PROGRAM AxisStop
VAR	
	
END_VAR

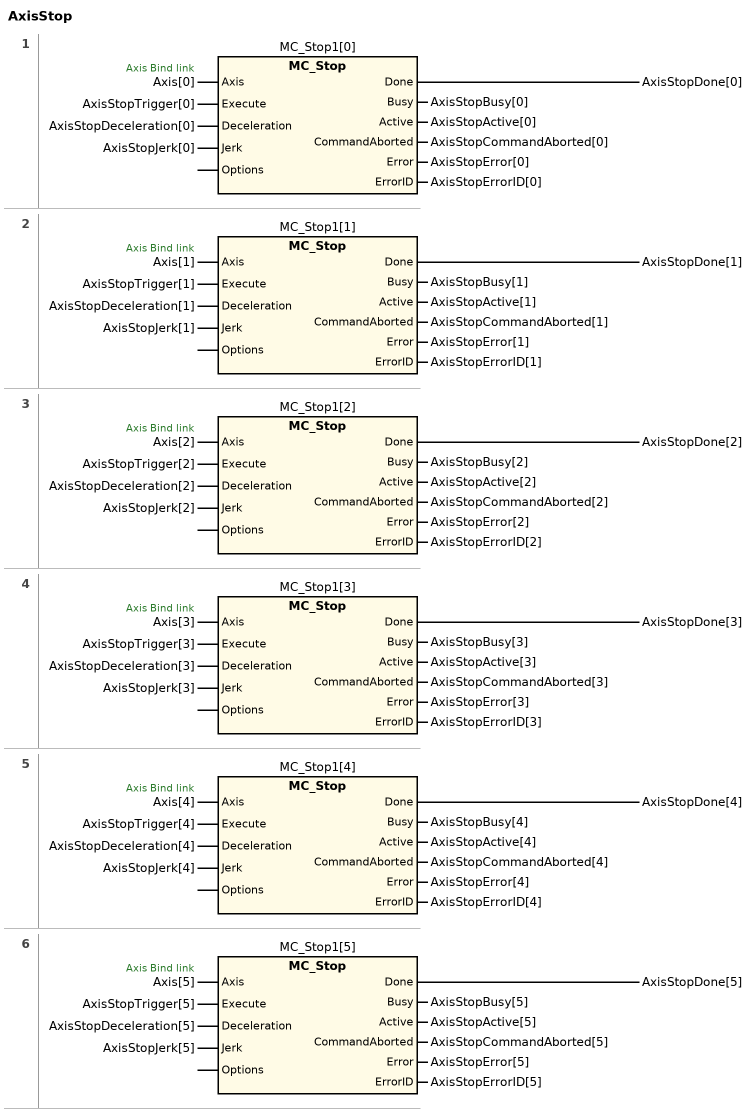
// NETWORK 1
//   MC_Stop1[0]: Axis Stop
//   Axis[0]: Axis Bind link
MC_Stop1[0](
    Axis := Axis[0],
    Execute := AxisStopTrigger[0],
    Deceleration := AxisStopDeceleration[0],
    Jerk := AxisStopJerk[0],
    Busy => AxisStopBusy[0],
    Active => AxisStopActive[0],
    CommandAborted => AxisStopCommandAborted[0],
    Error => AxisStopError[0],
    ErrorID => AxisStopErrorID[0]); // MC_Stop
AxisStopDone[0] := MC_Stop1[0].Done;

// NETWORK 2
//   MC_Stop1[1]: Axis Stop
//   Axis[1]: Axis Bind link
MC_Stop1[1](
    Axis := Axis[1],
    Execute := AxisStopTrigger[1],
    Deceleration := AxisStopDeceleration[1],
    Jerk := AxisStopJerk[1],
    Busy => AxisStopBusy[1],
    Active => AxisStopActive[1],
    CommandAborted => AxisStopCommandAborted[1],
    Error => AxisStopError[1],
    ErrorID => AxisStopErrorID[1]); // MC_Stop
AxisStopDone[1] := MC_Stop1[1].Done;

// NETWORK 3
//   MC_Stop1[2]: Axis Stop
//   Axis[2]: Axis Bind link
MC_Stop1[2](
    Axis := Axis[2],
    Execute := AxisStopTrigger[2],
    Deceleration := AxisStopDeceleration[2],
    Jerk := AxisStopJerk[2],
    Busy => AxisStopBusy[2],
    Active => AxisStopActive[2],
    CommandAborted => AxisStopCommandAborted[2],
    Error => AxisStopError[2],
    ErrorID => AxisStopErrorID[2]); // MC_Stop
AxisStopDone[2] := MC_Stop1[2].Done;

// NETWORK 4
//   MC_Stop1[3]: Axis Stop
//   Axis[3]: Axis Bind link
MC_Stop1[3](
    Axis := Axis[3],
    Execute := AxisStopTrigger[3],
    Deceleration := AxisStopDeceleration[3],
    Jerk := AxisStopJerk[3],
    Busy => AxisStopBusy[3],
    Active => AxisStopActive[3],
    CommandAborted => AxisStopCommandAborted[3],
    Error => AxisStopError[3],
    ErrorID => AxisStopErrorID[3]); // MC_Stop
AxisStopDone[3] := MC_Stop1[3].Done;

// NETWORK 5
//   MC_Stop1[4]: Axis Stop
//   Axis[4]: Axis Bind link
MC_Stop1[4](
    Axis := Axis[4],
    Execute := AxisStopTrigger[4],
    Deceleration := AxisStopDeceleration[4],
    Jerk := AxisStopJerk[4],
    Busy => AxisStopBusy[4],
    Active => AxisStopActive[4],
    CommandAborted => AxisStopCommandAborted[4],
    Error => AxisStopError[4],
    ErrorID => AxisStopErrorID[4]); // MC_Stop
AxisStopDone[4] := MC_Stop1[4].Done;

// NETWORK 6
//   MC_Stop1[5]: Axis Stop
//   Axis[5]: Axis Bind link
MC_Stop1[5](
    Axis := Axis[5],
    Execute := AxisStopTrigger[5],
    Deceleration := AxisStopDeceleration[5],
    Jerk := AxisStopJerk[5],
    Busy => AxisStopBusy[5],
    Active => AxisStopActive[5],
    CommandAborted => AxisStopCommandAborted[5],
    Error => AxisStopError[5],
    ErrorID => AxisStopErrorID[5]); // MC_Stop
AxisStopDone[5] := MC_Stop1[5].Done;

END_PROGRAM

(* stored: Version 1.1.0.1, ProductVersion 3.1.4018.5
   POU AxisStop: Id {b271ee6a-bc8e-43f9-90ca-9a15908bb5e1}, SpecialFunc None *)
